FUNCTION_BLOCK FB_GPWM
VAR_INPUT
	i_xEnable			: BOOL;
	i_udiTime			: UDINT;//PWM宽度时间，最小值为0，单位ms
	i_udiCycle			: UDINT;//PWM周期时间，最小值为1，单位ms
END_VAR
VAR_OUTPUT
	q_xOut				: BOOL;//占空比输出
END_VAR
VAR
	fbTon				: TON;
END_VAR

//数据保护
IF i_udiCycle < 1 THEN
	i_udiCycle := 1;
END_IF

IF i_udiTime > i_udiCycle THEN
	i_udiTime := i_udiCycle;
END_IF


//逻辑代码
IF i_xEnable THEN
	fbTon(IN:= TRUE, PT:= UDINT_TO_TIME(i_udiCycle));
	IF fbTon.Q THEN
		fbTon(IN:= FALSE);
	END_IF
	IF fbTon.ET <= UDINT_TO_TIME(i_udiTime) THEN
		q_xOut := TRUE;
	ELSE
		q_xOut := FALSE;
	END_IF
ELSE
	fbTon(IN:= FALSE);
	q_xOut := FALSE;
END_IF

END_FUNCTION_BLOCK

(* stored: Version 1.1.0.1, ProductVersion 3.1.4024.12
   POU FB_GPWM: Id {8bc82758-ebed-4e99-8faa-1c8ee63ebdc9}, SpecialFunc None *)
